FUNCTION_BLOCK Test_TEvent_AddEventHandler_ChecksInterfaceSupported EXTENDS TUnitTestbase
VAR
    TestEvent : TTestEvent;
    TestEventHandler : TUnsupportedEventHandler;
END_VAR

TestEvent.ClearEventHandlers().AddEventHandler(TestEventHandler); // should trigger an error message

Assertion.AssertEquals_UDINT(
    Expected := 0,
    Actual   := TestEvent.EventHandlers.Count,
    VariableName  := 'TestEvent.EventHandlers.Count');

_TestFinished := TRUE;

END_FUNCTION_BLOCK

(* stored: Version 1.1.0.1, ProductVersion 3.1.4024.4
   POU Test_TEvent_AddEventHandler_ChecksInterfaceSupported: Id {ac2ec9d9-50e6-4dbc-b579-c6a65abd5869}, SpecialFunc None *)
